(* CODESYS project TcL_Arrays.library
   Company: TwinCAT Libre
   Description: Basic functions for arrays.
   Version: 0.1
   DocFormat: reStructuredText
   Placeholder: TcL_Arrays
   Author: Ryan Severson
   Title: TcL_Arrays

Project tree, tasks and I/O mapping:
  DUTs/
    data type st_ArrayInfo
    data type st_ArrayInfoExt
    data type u_NumPointer
  Project Information/
    function F_GetCompany [ST]
    function F_GetTitle [ST]
    function F_GetVersion [ST]
  Version/
    global variables Global_Version
  function fn_ArrayAvg [ST]
  function fn_ArrayInfo [ST]
  function fn_ArrayMax [ST]
  function fn_ArrayMin [ST]
  function fn_ArraySize [ST]
  function fn_ArraySum [ST]
*)

// DUTs/st_ArrayInfo
//basic info for arrays
TYPE st_ArrayInfo :
STRUCT
	Size : DINT ; //number of elements in an array
	Sum : REAL;
	Average : REAL; //mean of the array
	Smallest : REAL; //smallest number in array
	Biggest : REAL; //largest number in array
	SmallestIndex : DINT; //position of smallest element
	BiggestIndex : DINT; //position of largest element
	Range : REAL; //difference between biggest and smallest
END_STRUCT
END_TYPE

// DUTs/st_ArrayInfoExt
//Extended array information
TYPE st_ArrayInfoExt EXTENDS st_ArrayInfo :
STRUCT
	Median : REAL; 
	Mode : REAL;
	StdDev : BOOL;
END_STRUCT
END_TYPE

// DUTs/u_NumPointer
//Union of all numerical types as pointers
TYPE u_NumPointer :
UNION
	pSINT : POINTER TO SINT; //8 bit
	pUSINT : POINTER TO USINT; //8 bit
	pINT : POINTER TO INT; //16 bit
	pUINT : POINTER TO UINT; //16 bit
	pDINT : POINTER TO DINT; //32 bit
	pUDINT : POINTER TO UDINT; //32 bit
	pLINT : POINTER TO LINT; //32 bit
	pULINT : POINTER TO ULINT; //32 bit
	pREAL : POINTER TO REAL; //32 bit
	pLREAL : POINTER TO LREAL; //64 bit
END_UNION
END_TYPE

// Version/Global_Version
{attribute 'TcGenerated'}
{attribute 'no-analysis'}
{attribute 'linkalways'}
// This function has been automatically generated from the project information.
VAR_GLOBAL CONSTANT
	{attribute 'const_non_replaced'}
	stLibVersion_TcL_Arrays : ST_LibVersion := (iMajor := 0, iMinor := 1, iBuild := 0, iRevision := 0, nFlags := 0, sVersion := '0.1');
END_VAR

// Project Information/F_GetCompany
// This function has been automatically generated from the project information.
{attribute 'signature_flag' := '1073741824'}
{attribute 'TcGenerated'}
{attribute 'no-analysis'}
FUNCTION F_GetCompany : WSTRING
VAR_INPUT
	
END_VAR

F_GetCompany := "TwinCAT Libre";

END_FUNCTION

// Project Information/F_GetTitle
// This function has been automatically generated from the project information.
{attribute 'signature_flag' := '1073741824'}
{attribute 'TcGenerated'}
{attribute 'no-analysis'}
FUNCTION F_GetTitle : WSTRING
VAR_INPUT
	
END_VAR

F_GetTitle := "TcL_Arrays";

END_FUNCTION

// Project Information/F_GetVersion
// This function has been automatically generated from the project information.
{attribute 'signature_flag' := '1073741824'}
{attribute 'TcGenerated'}
{attribute 'no-analysis'}
FUNCTION F_GetVersion : ST_LibVersion
VAR_INPUT
	
END_VAR

F_GetVersion.iMajor := 0;
F_GetVersion.iMinor := 1;
F_GetVersion.iBuild := 0;
F_GetVersion.iRevision := 0;

END_FUNCTION

// fn_ArrayAvg
(*
:Info: https://github.com/TwinCAT-Libre/
:Author: TwinCAT Libre

Version history:

+-------------+------------+----------+------------------------------------------+
|Date         | Version    | Author   | Remark                                   |
+=============+============+==========+==========================================+
|2022-04-15   | 0.1        | R.S.     | Initial Release                          |
+-------------+------------+----------+------------------------------------------+

Returns the average of all the elements in an array of any numerical type

*)

FUNCTION fn_ArrayAvg : REAL
VAR_INPUT 
	inArr : ANY; //Array to size
	inElem : ANY; //Any element in the array
END_VAR

VAR
	i : DINT := 0;
	size : DINT :=0; //number of elements in array
	pNum : u_NumPointer; //union of pointers of all numerical datatype	
END_VAR

size:= inArr.diSize/inElem.diSize;

CASE inElem.TypeClass OF
	__SYSTEM.TYPE_CLASS.TYPE_SINT:
		pNum.pSINT:=inArr.pValue;
		FOR i := 0 TO Size-1 DO
			fn_ArrayAvg := fn_ArrayAvg + pNum.pSINT[i];
		END_FOR;
		
	__SYSTEM.TYPE_CLASS.TYPE_USINT:
		pNum.pUSINT:=inArr.pValue;
		FOR i := 0 TO Size-1 DO
			fn_ArrayAvg := fn_ArrayAvg + pNum.pUSINT[i];
		END_FOR;
		
	__SYSTEM.TYPE_CLASS.TYPE_INT:
		pNum.pINT:=inArr.pValue;
		FOR i := 0 TO Size-1 DO
			fn_ArrayAvg := fn_ArrayAvg + pNum.pINT[i];
		END_FOR;

	__SYSTEM.TYPE_CLASS.TYPE_UINT:
		pNum.pUINT:=inArr.pValue;
		FOR i := 0 TO Size-1 DO
			fn_ArrayAvg := fn_ArrayAvg + pNum.pUINT[i];
		END_FOR;	
	
	__SYSTEM.TYPE_CLASS.TYPE_DINT:
		pNum.pDINT:=inArr.pValue;
		FOR i := 0 TO Size-1 DO
			fn_ArrayAvg := fn_ArrayAvg + DINT_TO_REAL(pNum.pDINT[i]);
		END_FOR;	
	
	__SYSTEM.TYPE_CLASS.TYPE_UDINT:
		pNum.pUDINT:=inArr.pValue;
		FOR i := 0 TO Size-1 DO
			fn_ArrayAvg := fn_ArrayAvg + UDINT_TO_REAL(pNum.pUDINT[i]);
		END_FOR;

	__SYSTEM.TYPE_CLASS.TYPE_LINT:
		pNum.pLINT:=inArr.pValue;
		FOR i := 0 TO Size-1 DO
			fn_ArrayAvg := fn_ArrayAvg + LINT_TO_REAL(pNum.pLINT[i]);
		END_FOR;		
		
	__SYSTEM.TYPE_CLASS.TYPE_ULINT:
		pNum.pULINT:=inArr.pValue;
		FOR i := 0 TO Size-1 DO
			fn_ArrayAvg := fn_ArrayAvg + ULINT_TO_REAL(pNum.pULINT[i]);
		END_FOR;		
		
	__SYSTEM.TYPE_CLASS.TYPE_REAL:
		pNum.pREAL:=inArr.pValue;
		FOR i := 0 TO Size-1 DO
			fn_ArrayAvg := fn_ArrayAvg + pNum.pREAL[i];
		END_FOR;

	__SYSTEM.TYPE_CLASS.TYPE_LREAL:	
		pNum.pLREAL:=inArr.pValue;
		FOR i := 0 TO Size-1 DO
			fn_ArrayAvg := fn_ArrayAvg + LREAL_TO_REAL(pNum.pLREAL[i]);
		END_FOR;		
ELSE
	fn_ArrayAvg :=0;
END_CASE;


fn_ArrayAvg := fn_ArrayAvg/DINT_TO_REAL(size);

END_FUNCTION

// fn_ArrayInfo
(*
:Info: https://github.com/TwinCAT-Libre/
:Author: TwinCAT Libre

Version history:

+-------------+------------+----------+------------------------------------------+
|Date         | Version    | Author   | Remark                                   |
+=============+============+==========+==========================================+
|2022-04-16   | 0.1        | R.S.     | Initial Release                          |
+-------------+------------+----------+------------------------------------------+

Returns the average,sum,size,range,limits from an array of any numerical type

*)

FUNCTION fn_ArrayInfo : st_ArrayInfo
VAR_INPUT 
	inArr : ANY; //Array to size
	inElem : ANY; //Any element in the array
END_VAR

VAR
	i : DINT := 0;
	pNum : u_NumPointer; //union of pointers of all numerical datatype	
END_VAR

fn_ArrayInfo.Size:= inArr.diSize/inElem.diSize;
fn_ArrayInfo.Smallest:=inArr.pValue[0];
fn_ArrayInfo.Biggest:=inArr.pValue[0];
fn_ArrayInfo.SmallestIndex:=0;
fn_ArrayInfo.BiggestIndex:=0;

CASE inElem.TypeClass OF
	
	__SYSTEM.TYPE_CLASS.TYPE_SINT:
		pNum.pSINT:=inArr.pValue;
		FOR i := 0 TO fn_ArrayInfo.Size-1 DO
			fn_ArrayInfo.Sum := fn_ArrayInfo.Sum + pNum.pSINT[i];
			IF pNum.pSINT[i] > fn_ArrayInfo.Biggest THEN
				fn_ArrayInfo.BiggestIndex:=i+1;
			END_IF
			IF pNum.pSINT[i] < fn_ArrayInfo.Smallest THEN
				fn_ArrayInfo.SmallestIndex:=i+1;
			END_IF				
				fn_ArrayInfo.Biggest:=MAX(fn_ArrayInfo.Biggest,pNum.pSINT[i]);
				fn_ArrayInfo.Smallest:=MIN(fn_ArrayInfo.Smallest,pNum.pSINT[i]);
		END_FOR;

	__SYSTEM.TYPE_CLASS.TYPE_USINT:
		pNum.pUSINT:=inArr.pValue;
		FOR i := 0 TO fn_ArrayInfo.Size-1 DO
			fn_ArrayInfo.Sum := fn_ArrayInfo.Sum + pNum.pUSINT[i];
			IF pNum.pUSINT[i] > fn_ArrayInfo.Biggest THEN
				fn_ArrayInfo.BiggestIndex:=i+1;
			END_IF
			IF pNum.pUSINT[i] < fn_ArrayInfo.Smallest THEN
				fn_ArrayInfo.SmallestIndex:=i+1;
			END_IF				
				fn_ArrayInfo.Biggest:=MAX(fn_ArrayInfo.Biggest,pNum.pUSINT[i]);
				fn_ArrayInfo.Smallest:=MIN(fn_ArrayInfo.Smallest,pNum.pUSINT[i]);
		END_FOR;
		
	__SYSTEM.TYPE_CLASS.TYPE_INT:
		pNum.pINT:=inArr.pValue;
		FOR i := 0 TO fn_ArrayInfo.Size-1 DO
			fn_ArrayInfo.Sum := fn_ArrayInfo.Sum + pNum.pINT[i];
			IF pNum.pINT[i] > fn_ArrayInfo.Biggest THEN
				fn_ArrayInfo.BiggestIndex:=i+1;
			END_IF
			IF pNum.pINT[i] < fn_ArrayInfo.Smallest THEN
				fn_ArrayInfo.SmallestIndex:=i+1;
			END_IF				
				fn_ArrayInfo.Biggest:=MAX(fn_ArrayInfo.Biggest,pNum.pINT[i]);
				fn_ArrayInfo.Smallest:=MIN(fn_ArrayInfo.Smallest,pNum.pINT[i]);
		END_FOR;
		
	__SYSTEM.TYPE_CLASS.TYPE_UINT:
		pNum.pUINT:=inArr.pValue;
		FOR i := 0 TO fn_ArrayInfo.Size-1 DO
			fn_ArrayInfo.Sum := fn_ArrayInfo.Sum + pNum.pUINT[i];
			IF pNum.pUINT[i] > fn_ArrayInfo.Biggest THEN
				fn_ArrayInfo.BiggestIndex:=i+1;
			END_IF
			IF pNum.pUINT[i] < fn_ArrayInfo.Smallest THEN
				fn_ArrayInfo.SmallestIndex:=i+1;
			END_IF				
				fn_ArrayInfo.Biggest:=MAX(fn_ArrayInfo.Biggest,pNum.pUINT[i]);
				fn_ArrayInfo.Smallest:=MIN(fn_ArrayInfo.Smallest,pNum.pUINT[i]);
		END_FOR;

	__SYSTEM.TYPE_CLASS.TYPE_DINT:
		pNum.pDINT:=inArr.pValue;
		FOR i := 0 TO fn_ArrayInfo.Size-1 DO
			fn_ArrayInfo.Sum := fn_ArrayInfo.Sum + DINT_TO_REAL(pNum.pDINT[i]);
			IF DINT_TO_REAL(pNum.pDINT[i]) > fn_ArrayInfo.Biggest THEN
				fn_ArrayInfo.BiggestIndex:=i+1;
			END_IF
			IF DINT_TO_REAL(pNum.pDINT[i]) < fn_ArrayInfo.Smallest THEN
				fn_ArrayInfo.SmallestIndex:=i+1;
			END_IF				
				fn_ArrayInfo.Biggest:=MAX(fn_ArrayInfo.Biggest,DINT_TO_REAL(pNum.pDINT[i]));
				fn_ArrayInfo.Smallest:=MIN(fn_ArrayInfo.Smallest,DINT_TO_REAL(pNum.pDINT[i]));
		END_FOR;

	__SYSTEM.TYPE_CLASS.TYPE_UDINT:
		pNum.pUDINT:=inArr.pValue;
		FOR i := 0 TO fn_ArrayInfo.Size-1 DO
			fn_ArrayInfo.Sum := fn_ArrayInfo.Sum + UDINT_TO_REAL(pNum.pUDINT[i]);
			IF UDINT_TO_REAL(pNum.pUDINT[i]) > fn_ArrayInfo.Biggest THEN
				fn_ArrayInfo.BiggestIndex:=i+1;
			END_IF
			IF UDINT_TO_REAL(pNum.pUDINT[i]) < fn_ArrayInfo.Smallest THEN
				fn_ArrayInfo.SmallestIndex:=i+1;
			END_IF				
				fn_ArrayInfo.Biggest:=MAX(fn_ArrayInfo.Biggest,UDINT_TO_REAL(pNum.pUDINT[i]));
				fn_ArrayInfo.Smallest:=MIN(fn_ArrayInfo.Smallest,UDINT_TO_REAL(pNum.pUDINT[i]));
		END_FOR;

	__SYSTEM.TYPE_CLASS.TYPE_LINT:
		pNum.pLINT:=inArr.pValue;
		FOR i := 0 TO fn_ArrayInfo.Size-1 DO
			fn_ArrayInfo.Sum := fn_ArrayInfo.Sum + LINT_TO_REAL(pNum.pLINT[i]);
			IF LINT_TO_REAL(pNum.pLINT[i]) > fn_ArrayInfo.Biggest THEN
				fn_ArrayInfo.BiggestIndex:=i+1;
			END_IF
			IF LINT_TO_REAL(pNum.pLINT[i]) < fn_ArrayInfo.Smallest THEN
				fn_ArrayInfo.SmallestIndex:=i+1;
			END_IF				
				fn_ArrayInfo.Biggest:=MAX(fn_ArrayInfo.Biggest,LINT_TO_REAL(pNum.pLINT[i]));
				fn_ArrayInfo.Smallest:=MIN(fn_ArrayInfo.Smallest,LINT_TO_REAL(pNum.pLINT[i])]);
		END_FOR;


	__SYSTEM.TYPE_CLASS.TYPE_ULINT:
		pNum.pULINT:=inArr.pValue;
		FOR i := 0 TO fn_ArrayInfo.Size-1 DO
			fn_ArrayInfo.Sum := fn_ArrayInfo.Sum + ULINT_TO_REAL(pNum.pULINT[i]);
			IF ULINT_TO_REAL(pNum.pULINT[i]) > fn_ArrayInfo.Biggest THEN
				fn_ArrayInfo.BiggestIndex:=i+1;
			END_IF
			IF ULINT_TO_REAL(pNum.pULINT[i]) < fn_ArrayInfo.Smallest THEN
				fn_ArrayInfo.SmallestIndex:=i+1;
			END_IF				
				fn_ArrayInfo.Biggest:=MAX(fn_ArrayInfo.Biggest,ULINT_TO_REAL(pNum.pULINT[i]));
				fn_ArrayInfo.Smallest:=MIN(fn_ArrayInfo.Smallest,ULINT_TO_REAL(pNum.pULINT[i]));
		END_FOR;
		
	__SYSTEM.TYPE_CLASS.TYPE_REAL:
		pNum.pREAL:=inArr.pValue;
		FOR i := 0 TO fn_ArrayInfo.Size-1 DO
			fn_ArrayInfo.Sum := fn_ArrayInfo.Sum + pNum.pREAL[i];
			IF pNum.pREAL[i] > fn_ArrayInfo.Biggest THEN
				fn_ArrayInfo.BiggestIndex:=i+1;
			END_IF
			IF pNum.pREAL[i] < fn_ArrayInfo.Smallest THEN
				fn_ArrayInfo.SmallestIndex:=i+1;
			END_IF				
				fn_ArrayInfo.Biggest:=MAX(fn_ArrayInfo.Biggest,pNum.pREAL[i]);
				fn_ArrayInfo.Smallest:=MIN(fn_ArrayInfo.Smallest,pNum.pREAL[i]);
		END_FOR;
	
	__SYSTEM.TYPE_CLASS.TYPE_LREAL:
		pNum.pLREAL:=inArr.pValue;
		FOR i := 0 TO fn_ArrayInfo.Size-1 DO
			fn_ArrayInfo.Sum := fn_ArrayInfo.Sum + pNum.pLREAL[i];
			IF pNum.pLREAL[i] > fn_ArrayInfo.Biggest THEN
				fn_ArrayInfo.BiggestIndex:=i+1;
			END_IF
			IF pNum.pLREAL[i] < fn_ArrayInfo.Smallest THEN
				fn_ArrayInfo.SmallestIndex:=i+1;
			END_IF				
				fn_ArrayInfo.Biggest:=MAX(fn_ArrayInfo.Biggest,pNum.pLREAL[i]);
				fn_ArrayInfo.Smallest:=MIN(fn_ArrayInfo.Smallest,pNum.pLREAL[i]);
		END_FOR;
ELSE
	fn_ArrayInfo.Sum :=0;
END_CASE;


fn_ArrayInfo.Average := fn_ArrayInfo.Sum/DINT_TO_REAL(fn_ArrayInfo.Size);
fn_ArrayInfo.Range := fn_ArrayInfo.Biggest - fn_ArrayInfo.Smallest;

END_FUNCTION

// fn_ArrayMax
(*
:Info: https://github.com/TwinCAT-Libre/
:Author: TwinCAT Libre

Version history:

+-------------+------------+----------+------------------------------------------+
|Date         | Version    | Author   | Remark                                   |
+=============+============+==========+==========================================+
|2022-04-12   | 0.1        | R.S.     | Initial Release                          |
+-------------+------------+----------+------------------------------------------+

Returns the largest value from an array of any numerical type

*)

FUNCTION fn_ArrayMax : REAL
VAR_INPUT 
	inArr : ANY; //Array to size
	inElem : ANY; //Any element in the array
END_VAR

VAR
	i : DINT := 0;
	size : DINT :=0; //number of elements in array
	pNum : u_NumPointer; //union of pointers of all numerical datatype
END_VAR

size:= inArr.diSize/inElem.diSize;
fn_ArrayMax:=inArr.pValue[0];
CASE inElem.TypeClass OF
	__SYSTEM.TYPE_CLASS.TYPE_SINT:
		pNum.pSINT:=inArr.pValue;
		FOR i := 0 TO Size-1 DO
			fn_ArrayMax:=Max(fn_ArrayMax,pNum.pSINT[i]);
		END_FOR;
		
	__SYSTEM.TYPE_CLASS.TYPE_USINT:
		pNum.pUSINT:=inArr.pValue;
		FOR i := 0 TO Size-1 DO
			fn_ArrayMax:=Max(fn_ArrayMax,pNum.pUSINT[i]);
		END_FOR;

	__SYSTEM.TYPE_CLASS.TYPE_INT:
		pNum.pINT:=inArr.pValue;
		FOR i := 0 TO Size-1 DO
			fn_ArrayMax:=Max(fn_ArrayMax,pNum.pINT[i]);
		END_FOR;	
		
	__SYSTEM.TYPE_CLASS.TYPE_DINT:
		pNum.pDINT:=inArr.pValue;
		FOR i := 0 TO Size-1 DO
			fn_ArrayMax:=Max(fn_ArrayMax,DINT_TO_REAL(pNum.pDINT[i]));
		END_FOR;

	__SYSTEM.TYPE_CLASS.TYPE_UDINT:
		pNum.pUDINT:=inArr.pValue;
		FOR i := 0 TO Size-1 DO
			fn_ArrayMax:=Max(fn_ArrayMax,UDINT_TO_REAL(pNum.pUDINT[i]));
		END_FOR;
		
	__SYSTEM.TYPE_CLASS.TYPE_LINT:
		pNum.pLINT:=inArr.pValue;
		FOR i := 0 TO Size-1 DO
			fn_ArrayMax:=Max(fn_ArrayMax,LINT_TO_REAL(pNum.pLINT[i]));
		END_FOR;
		
	__SYSTEM.TYPE_CLASS.TYPE_ULINT:
		pNum.pULINT:=inArr.pValue;
		FOR i := 0 TO Size-1 DO
			fn_ArrayMax:=Max(fn_ArrayMax,ULINT_TO_REAL(pNum.pULINT[i]));
		END_FOR;	

	__SYSTEM.TYPE_CLASS.TYPE_REAL:
		pNum.pREAL:=inArr.pValue;
		FOR i := 0 TO Size-1 DO
			fn_ArrayMax:=Max(fn_ArrayMax,pNum.pREAL[i]);
		END_FOR;		
	
	__SYSTEM.TYPE_CLASS.TYPE_LREAL:
		pNum.pLREAL:=inArr.pValue;
		FOR i := 0 TO Size-1 DO
			fn_ArrayMax:=Max(fn_ArrayMax,LREAL_TO_REAL(pNum.pLREAL[i]));
		END_FOR;		
	
ELSE
	fn_ArrayMax :=0;
END_CASE;

END_FUNCTION

// fn_ArrayMin
(*
:Info: https://github.com/TwinCAT-Libre/
:Author: TwinCAT Libre

Version history:

+-------------+------------+----------+------------------------------------------+
|Date         | Version    | Author   | Remark                                   |
+=============+============+==========+==========================================+
|2022-04-16   | 0.1        | R.S.     | Initial Release                          |
+-------------+------------+----------+------------------------------------------+

Returns the smallest value from an array of any numerical type

*)

FUNCTION fn_ArrayMin : REAL
VAR_INPUT 
	inArr : ANY; //Array to size
	inElem : ANY; //Any element in the array
END_VAR

VAR
	i : DINT := 0;
	size : DINT :=0; //number of elements in array
	pNum : u_NumPointer; //union of pointers of all numerical datatype
END_VAR

size:= inArr.diSize/inElem.diSize;
fn_ArrayMin:=inArr.pValue[0];
CASE inElem.TypeClass OF

	__SYSTEM.TYPE_CLASS.TYPE_SINT:
		pNum.pSINT:=inArr.pValue;
		FOR i := 0 TO Size-1 DO
			fn_ArrayMin:=MIN(fn_ArrayMin,pNum.pSINT[i]);
		END_FOR;
		
	__SYSTEM.TYPE_CLASS.TYPE_USINT:
		pNum.pUSINT:=inArr.pValue;
		FOR i := 0 TO Size-1 DO
			fn_ArrayMin:=MIN(fn_ArrayMin,pNum.pUSINT[i]);
		END_FOR;

	__SYSTEM.TYPE_CLASS.TYPE_INT:
		pNum.pINT:=inArr.pValue;
		FOR i := 0 TO Size-1 DO
			fn_ArrayMin:=MIN(fn_ArrayMin,pNum.pINT[i]);
		END_FOR;	
		
	__SYSTEM.TYPE_CLASS.TYPE_DINT:
		pNum.pDINT:=inArr.pValue;
		FOR i := 0 TO Size-1 DO
			fn_ArrayMin:=MIN(fn_ArrayMin,DINT_TO_REAL(pNum.pDINT[i]));
		END_FOR;

	__SYSTEM.TYPE_CLASS.TYPE_UDINT:
		pNum.pUDINT:=inArr.pValue;
		FOR i := 0 TO Size-1 DO
			fn_ArrayMin:=MIN(fn_ArrayMin,UDINT_TO_REAL(pNum.pUDINT[i]));
		END_FOR;
		
	__SYSTEM.TYPE_CLASS.TYPE_LINT:
		pNum.pLINT:=inArr.pValue;
		FOR i := 0 TO Size-1 DO
			fn_ArrayMin:=MIN(fn_ArrayMin,LINT_TO_REAL(pNum.pLINT[i]));
		END_FOR;
		
	__SYSTEM.TYPE_CLASS.TYPE_ULINT:
		pNum.pULINT:=inArr.pValue;
		FOR i := 0 TO Size-1 DO
			fn_ArrayMin:=MIN(fn_ArrayMin,ULINT_TO_REAL(pNum.pULINT[i]));
		END_FOR;	

	__SYSTEM.TYPE_CLASS.TYPE_REAL:
		pNum.pREAL:=inArr.pValue;
		FOR i := 0 TO Size-1 DO
			fn_ArrayMin:=MIN(fn_ArrayMin,pNum.pREAL[i]);
		END_FOR;		
	
	__SYSTEM.TYPE_CLASS.TYPE_LREAL:
		pNum.pLREAL:=inArr.pValue;
		FOR i := 0 TO Size-1 DO
			fn_ArrayMin:=MIN(fn_ArrayMin,LREAL_TO_REAL(pNum.pLREAL[i]));
		END_FOR;		
	
ELSE
	fn_ArrayMin :=0;
END_CASE;

END_FUNCTION

// fn_ArraySize
(*
:Info: https://github.com/TwinCAT-Libre/
:Author: TwinCAT Libre

Version history:

+-------------+------------+----------+------------------------------------------+
|Date         | Version    | Author   | Remark                                   |
+=============+============+==========+==========================================+
|2022-04-12   | 0.1        | R.S.     | Initial Release                          |
+-------------+------------+----------+------------------------------------------+

Returns the number of elements in an array of any type

*)

FUNCTION fn_ArraySize : UINT

VAR_INPUT 
	inArr : ANY; //Array to size
	inElem : ANY; //Any element in the array
END_VAR

fn_ArraySize:= DINT_TO_UINT(inArr.diSize/inElem.diSize);

END_FUNCTION

// fn_ArraySum
(*
:Info: https://github.com/TwinCAT-Libre/
:Author: TwinCAT Libre

Version history:

+-------------+------------+----------+------------------------------------------+
|Date         | Version    | Author   | Remark                                   |
+=============+============+==========+==========================================+
|2022-04-12   | 0.1        | R.S.     | Initial Release                          |
+-------------+------------+----------+------------------------------------------+

Returns the sum of elements in an array of any numerical type

*)

FUNCTION fn_ArraySum : REAL
VAR_INPUT 
	inArr : ANY; //Array to size
	inElem : ANY; //Any element in the array
END_VAR

VAR
	i : DINT := 0; //iterator
	size : DINT :=0; //number of elements in array
	pNum : u_NumPointer; //union of pointers of all numerical datatype
END_VAR

size:= inArr.diSize/inElem.diSize;

CASE inElem.TypeClass OF
	__SYSTEM.TYPE_CLASS.TYPE_SINT:
		pNum.pSINT:=inArr.pValue;
		FOR i := 0 TO Size-1 DO
			fn_ArraySum := fn_ArraySum + pNum.pSINT[i];
		END_FOR;
		
	__SYSTEM.TYPE_CLASS.TYPE_USINT:
		pNum.pUSINT:=inArr.pValue;
		FOR i := 0 TO Size-1 DO
			fn_ArraySum := fn_ArraySum + pNum.pUSINT[i];
		END_FOR;
		
	__SYSTEM.TYPE_CLASS.TYPE_INT:
		pNum.pINT:=inArr.pValue;
		FOR i := 0 TO Size-1 DO
			fn_ArraySum := fn_ArraySum + pNum.pINT[i];
		END_FOR;

	__SYSTEM.TYPE_CLASS.TYPE_UINT:
		pNum.pUINT:=inArr.pValue;
		FOR i := 0 TO Size-1 DO
			fn_ArraySum := fn_ArraySum + pNum.pUINT[i];
		END_FOR;	
	
	__SYSTEM.TYPE_CLASS.TYPE_DINT:
		pNum.pDINT:=inArr.pValue;
		FOR i := 0 TO Size-1 DO
			fn_ArraySum := fn_ArraySum + DINT_TO_REAL(pNum.pDINT[i]);
		END_FOR;	
	
	__SYSTEM.TYPE_CLASS.TYPE_UDINT:
		pNum.pUDINT:=inArr.pValue;
		FOR i := 0 TO Size-1 DO
			fn_ArraySum := fn_ArraySum + UDINT_TO_REAL(pNum.pUDINT[i]);
		END_FOR;

	__SYSTEM.TYPE_CLASS.TYPE_LINT:
		pNum.pLINT:=inArr.pValue;
		FOR i := 0 TO Size-1 DO
			fn_ArraySum := fn_ArraySum + LINT_TO_REAL(pNum.pLINT[i]);
		END_FOR;		
		
	__SYSTEM.TYPE_CLASS.TYPE_ULINT:
		pNum.pULINT:=inArr.pValue;
		FOR i := 0 TO Size-1 DO
			fn_ArraySum := fn_ArraySum + ULINT_TO_REAL(pNum.pULINT[i]);
		END_FOR;		
		
	__SYSTEM.TYPE_CLASS.TYPE_REAL:
		pNum.pREAL:=inArr.pValue;
		FOR i := 0 TO Size-1 DO
			fn_ArraySum := fn_ArraySum + pNum.pREAL[i];
		END_FOR;

	__SYSTEM.TYPE_CLASS.TYPE_LREAL:	
		pNum.pLREAL:=inArr.pValue;
		FOR i := 0 TO Size-1 DO
			fn_ArraySum := fn_ArraySum + LREAL_TO_REAL(pNum.pLREAL[i]);
		END_FOR;		
ELSE
	fn_ArraySum :=0;
END_CASE;

END_FUNCTION
